KUKA KRL program: panpick.src, panpick.dat

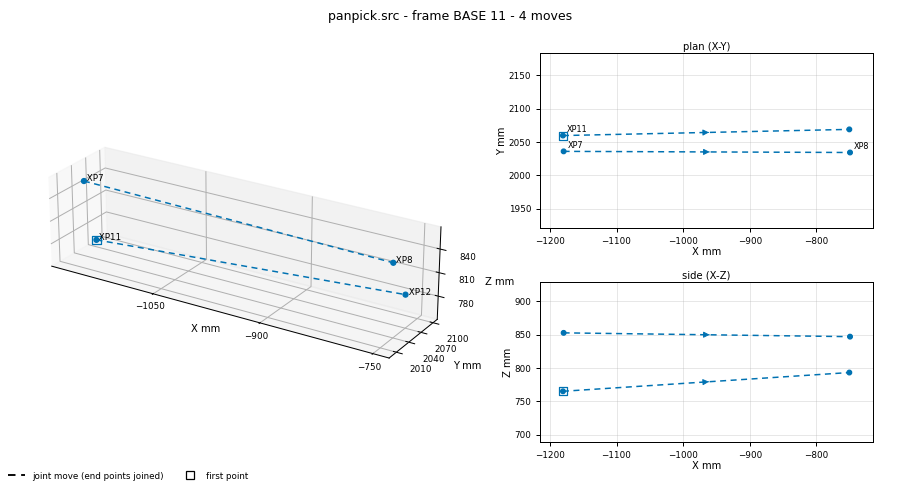
[picture p0: tool path of panpick.src in frame BASE 11, 4 of 13 moves have a stored position in this frame; points joined in program order, loops and branches not executed]
--- panpick.src ---
&ACCESS RVO1
&REL 3658
&PARAM EDITMASK = *
&PARAM TEMPLATE = C:\KRC\Roboter\Template\vorgabe
&PARAM DISKPATH = KRC:\R1\Program\Sub Programs
DEF panpick( )
;FOLD INI;%{PE}
  ;FOLD BASISTECH INI
    GLOBAL INTERRUPT DECL 3 WHEN $STOPMESS==TRUE DO IR_STOPM ( )
    INTERRUPT ON 3
    BAS (#INITMOV,0 )
  ;ENDFOLD (BASISTECH INI)
  ;FOLD USER INI
    ;Make your modifications here
INPICKER_Handler.DataToSend.command=0
 wait for (INPICKER_Handler.DataReceived.state==0)
REINTENTO=FALSE
;CILS_INIT()
  ;ENDFOLD (USER INI)
;ENDFOLD (INI)
;POS FOTO 1
XP03=$POS_ACT
PUNTOFOTO:
;FOLD PTP P03 Vel=100 % PDAT1 Tool[0] Base[0];%{PE}%R 8.3.48,%MKUKATPBASIS,%CMOVE,%VPTP,%P 1:PTP, 2:P03, 3:, 5:100, 7:PDAT1
$BWDSTART=FALSE
PDAT_ACT=PPDAT1
FDAT_ACT=FP03
BAS(#PTP_PARAMS,100)
PTP XP03
;ENDFOLD
INICIOFOTO:

;fold espera foto

 INPICKER_Handler.DataToSend.command=1
 wait for (INPICKER_Handler.DataReceived.state==30) or (INPICKER_Handler.DataReceived.state==-1)

 wait sec 0.5

 IF (INPICKER_Handler.DataReceived.state==-1) THEN
  ; wait for false
   IF (REINTENTO==FALSE) THEN

   REINTENTO=TRUE
   INPICKER_Handler.DataToSend.command=0
   wait for (INPICKER_Handler.DataReceived.state==0)
   GOTO INICIOFOTO

   ELSE

;FOTO NOK
;FOLD Fordtech.Tool_Req Tool Request: 1 ;%{PE}%MKUKATPUSER

Tool_Req (1)

;ENDFOLD
;FOLD Fordtech.Wait_Tool_Ready Wait Tool Ready: 1 ;%{PE}%MKUKATPUSER

Wait_Tool_Ready (1)

;ENDFOLD
BACKJUMP=TRUE
GOTO PEXIT

   ENDIF

ENDIF

;ENDFOLD

;EVALUA foto

IF (INPICKER_Handler.DataReceived.ObjectsGraspable>0)THEN

;FOLD CARGA FRAMEXP01
;FOTO OK
FRAMEAUX={X 0,Y 0,Z 0,A 0,B 0,C 0}
FRAMEAUX=INPICKER_Handler.DataReceived.PartsToGrasp0.Position
XP01.x=FRAMEAUX.x/10
XP01.y=(FRAMEAUX.y/10)-2
XP01.z=(FRAMEAUX.z/10)+7
XP01.a=(FRAMEAUX.a/10)+0.5
XP01.b=FRAMEAUX.b/10
XP01.c=FRAMEAUX.c/10
;ENDFOLD

;FOLD CARGA FRAME XP02
FRAMEAUX={X 0,Y 0,Z 0,A 0,B 0,C 0}
FRAMEAUX=INPICKER_Handler.DataReceived.PartsToGrasp0.PreGrasp0
XP02.x=FRAMEAUX.x/10
XP02.y=(FRAMEAUX.y/10)-2
XP02.z=(FRAMEAUX.z/10)+7
XP02.a=(FRAMEAUX.a/10)+0.5
XP02.b=FRAMEAUX.b/10
XP02.c=FRAMEAUX.c/10
;ENDFOLD

;FOLD OFFSET GIRADAS
IF ((INPICKER_Handler.DataReceived.PartsToGrasp0.Position.A > 890) AND (INPICKER_Handler.DataReceived.PartsToGrasp0.Position.A < 1100)) THEN

FRAMEAUX={X 0,Y 0,Z 0,A 0,B 0,C 0}
FRAMEAUX=INPICKER_Handler.DataReceived.PartsToGrasp0.Position
XP01.x=FRAMEAUX.x/10
XP01.y=(FRAMEAUX.y/10)-2
XP01.z=(FRAMEAUX.z/10)+7
XP01.a=(FRAMEAUX.a/10)+0.5
XP01.b=FRAMEAUX.b/10
XP01.c=FRAMEAUX.c/10

FRAMEAUX={X 0,Y 0,Z 0,A 0,B 0,C 0}
FRAMEAUX=INPICKER_Handler.DataReceived.PartsToGrasp0.PreGrasp0
XP02.x=FRAMEAUX.x/10
XP02.y=(FRAMEAUX.y/10)-2
XP02.z=(FRAMEAUX.z/10)+7
XP02.a=(FRAMEAUX.a/10)+0.5
XP02.b=FRAMEAUX.b/10
XP02.c=FRAMEAUX.c/10

ENDIF
;ENDFOLD


ELSE

IF (REINTENTO==FALSE) THEN
REINTENTO=TRUE
INPICKER_Handler.DataToSend.command=0
wait for (INPICKER_Handler.DataReceived.state==0)
GOTO INICIOFOTO
ENDIF

;FOTO NOK
;FOLD Fordtech.Tool_Req Tool Request: 1 ;%{PE}%MKUKATPUSER

Tool_Req (1)

;ENDFOLD
;FOLD Fordtech.Wait_Tool_Ready Wait Tool Ready: 1 ;%{PE}%MKUKATPUSER

Wait_Tool_Ready (1)

;ENDFOLD
BACKJUMP=TRUE
GOTO PEXIT

ENDIF

;Va a coger array

;Baja vel en arrays proximos a vallado
IF (posbat==11) THEN
;FOLD PTP P11 CONT Vel=100 % M2 Tool[5]:Gripper_empty Base[11];%{PE}%R 8.3.48,%MKUKATPBASIS,%CMOVE,%VPTP,%P 1:PTP, 2:P11, 3:C_DIS, 5:100, 7:M2
$BWDSTART=FALSE
PDAT_ACT=PM2
FDAT_ACT=FP11
BAS(#PTP_PARAMS,100)
PTP XP11 C_DIS
;ENDFOLD
ACT_OV=$OV_PRO
$OV_PRO=10
ENDIF

;Baja vel en arrays proximos a vallado
IF (posbat==12) THEN
;FOLD PTP P12 CONT Vel=100 % M2 Tool[5]:Gripper_empty Base[11];%{PE}%R 8.3.48,%MKUKATPBASIS,%CMOVE,%VPTP,%P 1:PTP, 2:P12, 3:C_DIS, 5:100, 7:M2
$BWDSTART=FALSE
PDAT_ACT=PM2
FDAT_ACT=FP12
BAS(#PTP_PARAMS,100)
PTP XP12 C_DIS
;ENDFOLD
ACT_OV=$OV_PRO
$OV_PRO=10
ENDIF

;FOLD PTP P02 CONT Vel=100 % PDAT2 Tool[5] Base[0];%{PE}%R 8.3.48,%MKUKATPBASIS,%CMOVE,%VPTP,%P 1:PTP, 2:P02, 3:C_DIS, 5:100, 7:PDAT2
$BWDSTART=FALSE
PDAT_ACT=PPDAT2
FDAT_ACT=FP02
BAS(#PTP_PARAMS,100)
PTP XP02 C_DIS
;ENDFOLD

;FOLD LIN P01 Vel=2 m/s CPDAT3 Tool[5] Base[0];%{PE}%R 8.3.48,%MKUKATPBASIS,%CMOVE,%VLIN,%P 1:LIN, 2:P01, 3:, 5:2, 7:CPDAT3
$BWDSTART=FALSE
LDAT_ACT=LCPDAT3
FDAT_ACT=FP01
BAS(#CP_PARAMS,2)
LIN XP01
;ENDFOLD
;halt
CIL_BAT_ACTIVO()

;Revisa sensores y si falta alguno abre y cierra la garra 1 vez
IF NOT (($IN[243] AND $IN[244] AND $IN[245] AND $IN[247])) THEN
  $OUT[243]=TRUE
  $OUT[244]=FALSE
  WAIT SEC 0.5
  $OUT[243]=FALSE
  $OUT[244]=TRUE
ENDIF

;Eleva batería 50mm
lin_rel {z 50}

$advance=0
;Revisa sensores de garra cerrados
;FOLD WAIT FOR ( IN 245 'CIL array closed S301B' );%{PE}%R 8.3.48,%MKUKATPBASIS,%CEXT_WAIT_FOR,%VEXT_WAIT_FOR,%P 2:, 4:, 5:$IN, 6:245, 7:CIL array closed S301B, 9:
WAIT FOR  ( $IN[245] )
;ENDFOLD
;FOLD WAIT FOR ( IN 247 'CIL array closed S302B' );%{PE}%R 8.3.48,%MKUKATPBASIS,%CEXT_WAIT_FOR,%VEXT_WAIT_FOR,%P 2:, 4:, 5:$IN, 6:247, 7:CIL array closed S302B, 9:
WAIT FOR  ( $IN[247] )
;ENDFOLD

PART_CHECK()

$advance=3
INPICKER_Handler.DataToSend.command=0

IF REINT_COGIDA==TRUE THEN
   lin_rel {z -40}
   CIL_BAT_REPOSO()
   PART_CHECK_OFF()
   lin_rel {z 100}
   wait for (INPICKER_Handler.DataReceived.state==0)
   GOTO PUNTOFOTO
ENDIF


;FOLD Fordtech.Tool_Req Tool Request: 2 ;%{PE}%MKUKATPUSER

Tool_Req (2)

;ENDFOLD
;FOLD Fordtech.Wait_Tool_Ready Wait Tool Ready: 2 ;%{PE}%MKUKATPUSER

Wait_Tool_Ready (2)

;ENDFOLD

;Fold guardamos posicion para carton
IF (POSBAT==12) THEN
   ;IF ($POS_ACT.x>-920) AND ($POS_ACT.x<-690) THEN
   IF ($POS_ACT.x>-970) AND ($POS_ACT.x<-640) THEN
      BASE_DATA[14].x=$POS_ACT.x
   ENDIF
;   IF ($POS_ACT.y<2257) AND ($POS_ACT.y>2057) THEN
   IF ($POS_ACT.y<2307) AND ($POS_ACT.y>2007) THEN
      BASE_DATA[14].y=$POS_ACT.y
   ENDIF
;BASE_DATA[14].z=$POS_ACT.z
ENDIF
;ENDFOLD


;fold P04

FRAMEAUX={X 0,Y 0,Z 0,A 0,B 0,C 0}
XP04=FRAMEAUX
XP04.x=XP02.x
XP04.y=XP02.y
XP04.z=(XP02.z)+110
XP04.a=XP02.a
XP04.b=XP02.b
XP04.c=XP02.c

;ENDFOLD

;FOLD PTP p04 CONT Vel=100 % PDAT4 Tool[8]:Gripper_array Base[0];%{PE}%R 8.3.48,%MKUKATPBASIS,%CMOVE,%VPTP,%P 1:PTP, 2:p04, 3:C_DIS, 5:100, 7:PDAT4
$BWDSTART=FALSE
PDAT_ACT=PPDAT4
FDAT_ACT=Fp04
BAS(#PTP_PARAMS,100)
PTP Xp04 C_DIS
;ENDFOLD

IF (posbat==11) THEN
;FOLD PTP P7 CONT Vel=100 % H Tool[5]:Gripper_empty Base[11];%{PE}%R 8.3.48,%MKUKATPBASIS,%CMOVE,%VPTP,%P 1:PTP, 2:P7, 3:C_DIS, 5:100, 7:H
$BWDSTART=FALSE
PDAT_ACT=PH
FDAT_ACT=FP7
BAS(#PTP_PARAMS,100)
PTP XP7 C_DIS
;ENDFOLD
$OV_PRO=ACT_OV
ENDIF

IF (posbat==12) THEN
;FOLD PTP P8 CONT Vel=100 % H Tool[5]:Gripper_empty Base[11];%{PE}%R 8.3.48,%MKUKATPBASIS,%CMOVE,%VPTP,%P 1:PTP, 2:P8, 3:C_DIS, 5:100, 7:H
$BWDSTART=FALSE
PDAT_ACT=PH
FDAT_ACT=FP8
BAS(#PTP_PARAMS,100)
PTP XP8 C_DIS
;ENDFOLD
$OV_PRO=ACT_OV
ENDIF

;FOLD SYN OUT 41 'Job Ready 1' State=TRUE at START Delay=0 ms;%{PE}%R 8.3.48,%MKUKATPBASIS,%COUT,%VSYNOUT,%P 2:41, 3:Job Ready 1, 5:TRUE, 7:0, 9:0, 12:0
TRIGGER WHEN DISTANCE=0 DELAY=0 DO $OUT[41]=TRUE
;ENDFOLD
BAT_MONITOR=TRUE

;FOLD PTP P4 CONT Vel=90 % M2 Tool[8]:Gripper_array Base[0];%{PE}%R 8.3.48,%MKUKATPBASIS,%CMOVE,%VPTP,%P 1:PTP, 2:P4, 3:C_DIS, 5:90, 7:M2
$BWDSTART=FALSE
PDAT_ACT=PM2
FDAT_ACT=FP4
BAS(#PTP_PARAMS,90)
PTP XP4 C_DIS
;ENDFOLD
;FOLD SYN OUT 17 'Area Release 1' State=TRUE at START Delay=0 ms;%{PE}%R 8.3.48,%MKUKATPBASIS,%COUT,%VSYNOUT,%P 2:17, 3:Area Release 1, 5:TRUE, 7:0, 9:0, 12:0
TRIGGER WHEN DISTANCE=0 DELAY=0 DO $OUT[17]=TRUE
;ENDFOLD
;FOLD PTP P6 CONT Vel=100 % PDAT6 Tool[8]:Gripper_array Base[0];%{PE}%R 8.3.48,%MKUKATPBASIS,%CMOVE,%VPTP,%P 1:PTP, 2:P6, 3:C_DIS, 5:100, 7:PDAT6
$BWDSTART=FALSE
PDAT_ACT=PPDAT6
FDAT_ACT=FP6
BAS(#PTP_PARAMS,100)
PTP XP6 C_DIS
;ENDFOLD

PEXIT:
END

--- panpick.dat ---
&ACCESS RVO1
&REL 3658
&PARAM EDITMASK = *
&PARAM TEMPLATE = C:\KRC\Roboter\Template\vorgabe
&PARAM DISKPATH = KRC:\R1\Program\Sub Programs
DEFDAT  panpick
;FOLD EXTERNAL DECLARATIONS;%{PE}%MKUKATPBASIS,%CEXT,%VCOMMON,%P
;FOLD BASISTECH EXT;%{PE}%MKUKATPBASIS,%CEXT,%VEXT,%P
EXT  BAS (BAS_COMMAND  :IN,REAL  :IN )
DECL INT SUCCESS
;ENDFOLD (BASISTECH EXT)
;FOLD USER EXT;%{E}%MKUKATPUSER,%CEXT,%VEXT,%P
;Make your modifications here

;ENDFOLD (USER EXT)
;ENDFOLD (EXTERNAL DECLARATIONS)
DECL E6POS XP01={X -743.900,Y 2175.00,Z 682.200,A 270.200,B 359.900,C 179.600}
DECL FDAT FP01={TOOL_NO 5,BASE_NO 0,IPO_FRAME #BASE,POINT2[] " "}
DECL PDAT PPDAT01={VEL 100.000,ACC 100.000,APO_DIST 500.000,APO_MODE #CDIS,GEAR_JERK 100.000,EXAX_IGN 0}
DECL MODULEPARAM_T LAST_TP_PARAMS={PARAMS[] "Kuka.VelocityFieldEnabled=True; Kuka.ColDetectFieldEnabled=True; Kuka.MovementParameterFieldEnabled=True; Kuka.IsAngleEnabled=False; Kuka.PointName=P02; Kuka.FrameData.base_no=0; Kuka.FrameData.tool_no=5; Kuka.FrameData.ipo_frame=#BASE; Kuka.isglobalpoint=False; Kuka.MoveDataPtpName=PDAT02; Kuka.MovementDataPdat.apo_mode=#CDIS; Kuka.MovementDataPdat.apo_dist=500; Kuka.MovementData.vel=2; Kuka.MovementData.acc=100; Kuka.MovementData.exax_ign=0; Kuka.VelocityPtp=100; Kuka.BlendingEnabled=False; Kuka.APXEnabled=False; Kuka.CurrentCDSetIndex=0; Kuka.FrameData.point2=; Kuka.MoveDataName=CPDAT2; Kuka.MovementData.cb={AUX_PT {ORI #CONSIDER,E1 #CONSIDER,E2 #CONSIDER,E3 #CONSIDER,E4 #CONSIDER,E5 #CONSIDER,E6 #CONSIDER},TARGET_PT {ORI #INTERPOLATE,E1 #INTERPOLATE,E2 #INTERPOLATE,E3 #INTERPOLATE,E4 #INTERPOLATE,E5 #INTERPOLATE,E6 #INTERPOLATE}}; Kuka.MovementData.apo_fac=50; Kuka.MovementData.apo_dist=500; Kuka.MovementData.axis_acc=100; Kuka.MovementData.axis_vel=100; Kuka.MovementData.circ_typ=#BASE; Kuka.MovementData.jerk_fac=50; Kuka.MovementData.ori_typ=#VAR; Kuka.VelocityPath=2                          "}
DECL E6POS XP02={X -743.600,Y 2175.10,Z 732.200,A 270.200,B 359.900,C 179.600}
DECL FDAT FP02={TOOL_NO 5,BASE_NO 0,IPO_FRAME #BASE,POINT2[] " "}
DECL PDAT PPDAT02={VEL 100.000,ACC 100.000,APO_DIST 500.000,APO_MODE #CDIS,GEAR_JERK 100.000,EXAX_IGN 0}
DECL LDAT LCPDAT1={VEL 2.00000,ACC 100.000,APO_DIST 500.000,APO_FAC 50.0000,AXIS_VEL 100.000,AXIS_ACC 100.000,ORI_TYP #VAR,CIRC_TYP #BASE,JERK_FAC 50.0000,GEAR_JERK 100.000,EXAX_IGN 0,CB {AUX_PT {ORI #CONSIDER,E1 #CONSIDER,E2 #CONSIDER,E3 #CONSIDER,E4 #CONSIDER,E5 #CONSIDER,E6 #CONSIDER},TARGET_PT {ORI #INTERPOLATE,E1 #INTERPOLATE,E2 #INTERPOLATE,E3 #INTERPOLATE,E4 #INTERPOLATE,E5 #INTERPOLATE,E6 #INTERPOLATE}}}
DECL E6POS XP03={X -523.662537,Y 1683.77332,Z 1415.68750,A -86.9886169,B 22.0730648,C -178.936188,S 'B0110',T 'B00011011',E1 0.0,E2 0.0,E3 0.0,E4 0.0,E5 0.0,E6 0.0}
DECL FDAT FP03={TOOL_NO 0,BASE_NO 0,IPO_FRAME #BASE,POINT2[] " "}
DECL PDAT PPDAT03={VEL 100.000,ACC 100.000,APO_DIST 500.000,APO_MODE #CDIS,GEAR_JERK 100.000,EXAX_IGN 0}
DECL E6POS XP04={X -743.600,Y 2175.10,Z 842.200,A 270.200,B 359.900,C 179.600}
DECL FDAT FP04={TOOL_NO 8,BASE_NO 0,IPO_FRAME #BASE,POINT2[] " ",TQ_STATE FALSE}
DECL PDAT PPDAT04={VEL 100.000,ACC 100.000,APO_DIST 500.000,APO_MODE #CDIS,GEAR_JERK 100.000,EXAX_IGN 0}
DECL E6POS XP1={X 2856.00,Y 12860.0,Z 6727.00,A 2708.00,B 8.00000,C 1797.00}
DECL E6POS XP2={X 2856.00,Y 12860.0,Z 6727.00,A 2708.00,B 8.00000,C 1797.00}
DECL E6POS XP3={X 2856.00,Y 12860.0,Z 6727.00,A 2708.00,B 8.00000,C 1797.00}
DECL E6POS XP05={X 284.000,Y 1258.50,Z 983.400,A 271.300,B 0.800000,C 179.700,S 0,T 0,E1 0.0,E2 0.0,E3 0.0,E4 0.0,E5 0.0,E6 0.0}
DECL FDAT FP05={TOOL_NO 5,BASE_NO 0,IPO_FRAME #BASE,POINT2[] " "}
DECL PDAT PPDAT05={VEL 100.000,ACC 100.000,APO_DIST 500.000,APO_MODE #CDIS,GEAR_JERK 100.000,EXAX_IGN 0}
DECL LDAT LCPDAT2={VEL 2.00000,ACC 100.000,APO_DIST 500.000,APO_FAC 50.0000,AXIS_VEL 100.000,AXIS_ACC 100.000,ORI_TYP #VAR,CIRC_TYP #BASE,JERK_FAC 50.0000,GEAR_JERK 100.000,EXAX_IGN 0,CB {AUX_PT {ORI #CONSIDER,E1 #CONSIDER,E2 #CONSIDER,E3 #CONSIDER,E4 #CONSIDER,E5 #CONSIDER,E6 #CONSIDER},TARGET_PT {ORI #INTERPOLATE,E1 #INTERPOLATE,E2 #INTERPOLATE,E3 #INTERPOLATE,E4 #INTERPOLATE,E5 #INTERPOLATE,E6 #INTERPOLATE}}}
DECL BASIS_SUGG_T LAST_BASIS={POINT1[] "P8                      ",POINT2[] "P8                      ",CP_PARAMS[] "CPDAT0                  ",PTP_PARAMS[] "PDAT7                   ",CONT[] "                        ",CP_VEL[] "2.0                     ",PTP_VEL[] "100                     ",SYNC_PARAMS[] "SYNCDAT                 ",SPL_NAME[] "S0                      ",A_PARAMS[] "ADAT0                   "}
DECL PDAT PPDAT1={VEL 100.000,ACC 100.000,APO_DIST 100.000,GEAR_JERK 50.0000,EXAX_IGN 0}
DECL PDAT PPDAT2={VEL 100.000,ACC 100.000,APO_DIST 100.000,APO_MODE #CDIS,GEAR_JERK 50.0000,EXAX_IGN 0}
DECL LDAT LCPDAT3={VEL 2.00000,ACC 100.000,APO_DIST 100.000,APO_FAC 50.0000,AXIS_VEL 100.000,AXIS_ACC 100.000,ORI_TYP #VAR,CIRC_TYP #BASE,JERK_FAC 50.0000,GEAR_JERK 50.0000,EXAX_IGN 0}
DECL LDAT LCPDAT4={VEL 2.00000,ACC 100.000,APO_DIST 100.000,APO_FAC 50.0000,AXIS_VEL 100.000,AXIS_ACC 100.000,ORI_TYP #VAR,CIRC_TYP #BASE,JERK_FAC 50.0000,GEAR_JERK 50.0000,EXAX_IGN 0}
DECL E6POS XP4={X 290.951233,Y 816.177124,Z 1275.55042,A -86.9976196,B 22.0779018,C -179.006119,S 6,T 27,E1 0.0,E2 0.0,E3 0.0,E4 0.0,E5 0.0,E6 0.0}
DECL FDAT FP4={TOOL_NO 8,BASE_NO 0,IPO_FRAME #BASE,POINT2[] " ",TQ_STATE FALSE}
DECL PDAT PPDAT3={VEL 100.000,ACC 100.000,APO_DIST 100.000,APO_MODE #CDIS,GEAR_JERK 50.0000,EXAX_IGN 0}
DECL PDAT PPDAT4={VEL 100.000,ACC 100.000,APO_DIST 100.000,APO_MODE #CDIS,GEAR_JERK 50.0000,EXAX_IGN 0}
DECL E6POS XP5={X 442.124359,Y -682.465210,Z 1416.05603,A -171.206314,B 14.8656197,C -154.747955,S 6,T 26,E1 0.0,E2 0.0,E3 0.0,E4 0.0,E5 0.0,E6 0.0}
DECL FDAT FP5={TOOL_NO 8,BASE_NO 0,IPO_FRAME #BASE,POINT2[] " ",TQ_STATE FALSE}
DECL PDAT PPDAT5={VEL 100.000,ACC 100.000,APO_DIST 100.000,APO_MODE #CDIS,GEAR_JERK 50.0000,EXAX_IGN 0}
DECL E6POS XP6={X 476.912292,Y -740.186951,Z 1393.23120,A -161.119644,B 4.43573570,C -171.398254,S 6,T 26,E1 0.0,E2 0.0,E3 0.0,E4 0.0,E5 0.0,E6 0.0}
DECL FDAT FP6={TOOL_NO 8,BASE_NO 0,IPO_FRAME #BASE,POINT2[] " ",TQ_STATE FALSE}
DECL PDAT PPDAT6={VEL 100.000,ACC 100.000,APO_DIST 100.000,APO_MODE #CDIS,GEAR_JERK 50.0000,EXAX_IGN 0}
DECL E6POS XP11={X -1180.39600,Y 2059.83276,Z 765.081604,A -88.4982,B 3.76465464,C -179.963882,S 6,T 27,E1 0.0,E2 0.0,E3 0.0,E4 0.0,E5 0.0,E6 0.0}
DECL FDAT FP11={TOOL_NO 5,BASE_NO 11,IPO_FRAME #BASE,POINT2[] " ",TQ_STATE FALSE}
DECL PDAT PM2={VEL 100.000,ACC 70.0000,APO_DIST 300.000,APO_MODE #CDIS,GEAR_JERK 50.0000,EXAX_IGN 0}
DECL PDAT PM3={VEL 100.000,ACC 70.0000,APO_DIST 300.000,APO_MODE #CDIS,GEAR_JERK 50.0000,EXAX_IGN 0}
DECL E6POS XP12={X -750.455750,Y 2069.09058,Z 793.223267,A -88.0968246,B 5.56702805,C -179.655121,S 6,T 27,E1 0.0,E2 0.0,E3 0.0,E4 0.0,E5 0.0,E6 0.0}
DECL FDAT FP12={TOOL_NO 5,BASE_NO 11,IPO_FRAME #BASE,POINT2[] " ",TQ_STATE FALSE}
DECL PDAT PM4={VEL 100.000,ACC 70.0000,APO_DIST 300.000,APO_MODE #CDIS,GEAR_JERK 50.0000,EXAX_IGN 0}
DECL E6POS XP0={X -1180.39600,Y 2059.83276,Z 765.081604,A -88.4982,B 3.76465464,C -179.963882,S 6,T 27,E1 0.0,E2 0.0,E3 0.0,E4 0.0,E5 0.0,E6 0.0}
DECL FDAT FP0={TOOL_NO 5,BASE_NO 11,IPO_FRAME #BASE,POINT2[] " ",TQ_STATE FALSE}
DECL PDAT PM5={VEL 100.000,ACC 70.0000,APO_DIST 300.000,APO_MODE #CDIS,GEAR_JERK 50.0000,EXAX_IGN 0}
DECL E6POS XP7={X -1179.40,Y 2036.10010,Z 852.800,A -88.3999939,B -0.399993837,C 179.200,S 6,T 27,E1 0.0,E2 0.0,E3 0.0,E4 0.0,E5 0.0,E6 0.0}
DECL FDAT FP7={TOOL_NO 5,BASE_NO 11,IPO_FRAME #BASE,POINT2[] " ",TQ_STATE FALSE}
DECL PDAT PH={VEL 100.000,ACC 100.000,APO_DIST 300.000,APO_MODE #CDIS,GEAR_JERK 50.0000,EXAX_IGN 0}
DECL PDAT PPDAT7={VEL 100.000,ACC 100.000,APO_DIST 100.000,GEAR_JERK 50.0000,EXAX_IGN 0}
DECL E6POS XP8={X -749.400,Y 2034.39990,Z 847.100,A -88.2000122,B -0.499999970,C 179.600,S 6,T 27,E1 0.0,E2 0.0,E3 0.0,E4 0.0,E5 0.0,E6 0.0}
DECL FDAT FP8={TOOL_NO 5,BASE_NO 11,IPO_FRAME #BASE,POINT2[] " ",TQ_STATE FALSE}
ENDDAT
